TYPE ST_GantryXYZ_Config :
    STRUCT
	CuttingHeightZ : REAL;
	CuttingSpeedX :REAL;
	CuttingSpeedY :REAL;
	CuttingSpeedZ :REAL;
	IdleTime :REAL;
	PanelFrontLength : REAL;
	PanelFrontWidht : REAL;
	PanelHeight : REAL;
	ProgramIdRequested : REAL;
	RailHeightCorrection :REAL;
	RapidSpeedX :REAL;
	RapidSpeedY :REAL;
	RapidSpeedZ :REAL;
	ToolOverpass :REAL;
    END_STRUCT
END_TYPE

(* stored: Version 1.1.0.1, ProductVersion 3.1.4024.15
   DUT ST_GantryXYZ_Config: Id {9175d3d8-e623-4395-a625-175ecc53cdb9} *)
